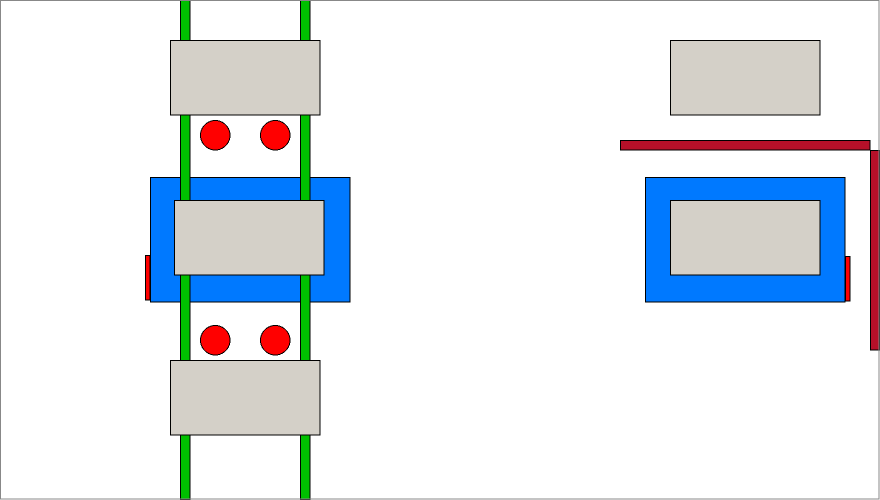
VISUALIZATION vTransporterSequence_1  // 880x500
VAR_IN_OUT
	iWorkStep	: INT;
END_VAR
    Rectangle (150,177 200x125)
    Rectangle (645,177 200x125)
    Rectangle (300,0 10x500)
    Rectangle (180,0 10x500)
    Rectangle (170,40 150x75)
    Rectangle (170,360 150x75)
    Rectangle (670,200 150x75)
    Rectangle (174,200 150x75)
    Rectangle (670,40 150x75), invisible if: NOT iWorkStep=20
    Ellipse (200,120 30x30)
    Ellipse (260,120 30x30)
    Ellipse (260,325 30x30)
    Ellipse (200,325 30x30)
    Rectangle (870,150 10x200)
    Rectangle (620,140 250x10)
    Rectangle (845,256 5x45)
    Rectangle (145,255 5x45)
END_VISUALIZATION

(* stored: Version 1.1.0.1, ProductVersion 3.1.4024.13
   Visu vTransporterSequence_1: Id {31f5ca45-8356-4f21-814b-cc72ec0ba200} *)
